{attribute 'qualified_only'}
{attribute 'strict'}
{attribute 'to_string'}
TYPE SerialFlowControl :
(
	None := 0,
	XonXoff,
	RtsCts,
	DsrDts
);
END_TYPE

(* stored: Version 1.1.0.1, ProductVersion 3.1.4024.3
   DUT SerialFlowControl: Id {0692c14f-e4b2-4d54-b2da-0bd8d92552e0} *)
